// TIA Portal V17 export
// export: Created 2025-12-08T12:10:26.7684921Z, ExportSetting WithDefaults, DisplayName Totally Integrated Automation Portal, DisplayVersion V17 Update 7, DisplayName TIA Portal Openness, DisplayVersion V17 Update 7, DisplayName TIA Portal Version Control Interface, DisplayVersion V17, DisplayName SINAMICS Startdrive Advanced, DisplayVersion V17 SP2, DisplayName SINAMICS DCC, DisplayVersion V17 Update 1, DisplayName SINAMICS Startdrive G110M, G120, G120C, G120D, G120P, G115D, DisplayVersion V17 SP2, DisplayName SINAMICS Startdrive G130, G150, S120, S150, SINAMICS MV, S210, DisplayVersion V17 SP2, DisplayName STEP 7 Professional, DisplayVersion V17 Update 7, DisplayName STEP 7 Safety, DisplayVersion V17 Update 6, DisplayName WinCC Advanced, DisplayVersion V17 Update 7
FUNCTION "ADDITION" : Void   // FC1, LAD
{ S7_Optimized_Access := 'TRUE' }
VERSION : 0.1
// stored: AutoNumber true, IsIECCheckEnabled false, SetENOAutomatically false, UDAEnableTagReadback false
   VAR_INPUT
      "A" : Int;
      "B" : Int;
      C : Int;
   END_VAR
   VAR_OUTPUT
      RESULT : Int;
   END_VAR
   VAR_TEMP
      OUT : Int;
   END_VAR
BEGIN

REGION Network 1
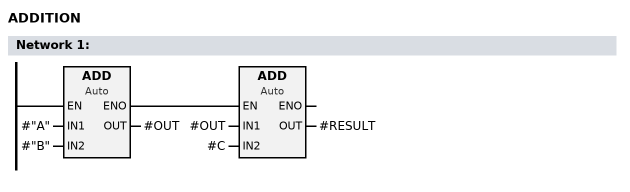
   RUNG wire#powerrail
      Add(in1 := #"A", in2 := #"B", out => #OUT)
      Add(in1 := #OUT, in2 := #C, out => #RESULT)
   END_RUNG
   // the same network as SCL:
   #OUT := #"A" + #"B";
   #RESULT := #OUT + #C;
END_REGION
END_FUNCTION
